// TIA Portal project "Bekletme_Kesmesi_Uygulaması_V1" (V16)
// Vorlageprojekt für das Buch mit Zielsystem S7-1200

(* hardware
DEVICE "S7-1200-Station_1"  S7-1200 Station
   slot 0: "Baugruppenträger_0"  Rack  V1.0
   slot 1: "PLC_1"  CPU 1214C DC/DC/DC  6ES7 214-1AG40-0XB0  V4.4
*)

// ===== PLC "PLC_1"  CPU 1214C DC/DC/DC =====

VAR_GLOBAL   // PLC tag table "Standard-Variablentabelle"
   "Sistem_Start_Mem." AT %M10.0 : Bool;
   "Kenar_Darbesi_1" AT %M20.0 : Bool;
   "Alarm" AT %M30.0 : Bool;
   "Kenar_Darbesi_2" AT %M20.1 : Bool;
   "Tag_1" AT %MW32 : Word;
   "Tag_2" AT %MW34 : Int;
END_VAR

VAR_GLOBAL   // PLC tag table "İnput"
   "Start_But" AT %I0.0 : Bool;
   "Stop_But" AT %I0.1 : Bool;
   "Sürücü_Geri_Sensörü" AT %I0.2 : Bool;
   "Sürücü_İleri_Sensörü" AT %I0.3 : Bool;
   "Optik_Sensör" AT %I0.4 : Bool;
   "Konveyör_Hız_Ayarı" AT %IW30 : Int;
END_VAR

VAR_GLOBAL   // PLC tag table "Output"
   "Sürücü" AT %Q0.0 : Bool;
   "Uyarı_Lambası" AT %Q0.1 : Bool;
   "Konveyör_1" AT %QW30 : Int;
   "Konveyör_2" AT %QW32 : Int;
END_VAR

FUNCTION "MHJ-PLC-Lab-Function-S71200" : Void   // FC9000, SCL
{ S7_Optimized_Access := 'TRUE' }
VERSION : 0.1
   VAR_TEMP
      rdTimeReturn : Int;
      outputTime : DTL;
      SyncVal : Byte;
      forVal : Int;
      forVal_2 : Int;
      Value : Byte;
   END_VAR
   VAR CONSTANT
      CompVal : Byte := 16#34;
      Value_01 : Byte := 16#11;
      Value_01_DW : DWord := 16#A165_D992;
      Value_02_DW : DWord := 16#58BE_4401;
   END_VAR
BEGIN

   #Value:=PEEK(area := 16#82,
        dbNumber := 0,
        byteOffset := 511);
   #Value := #Value + 1;

   POKE(area := 16#82,
        dbNumber := 0,
        byteOffset := 511,
        value := #Value);

   POKE(area:=16#81,
        dbNumber:=0,
        byteOffset:=1016,
        value:=#Value_01_DW);
   POKE(area := 16#81,
        dbNumber := 0,
        byteOffset := 1020,
        value := #Value_02_DW);

   POKE(area := 16#81,
        dbNumber := 0,
        byteOffset := 511,
        value := B#16#00);

   FOR #forVal := 0 TO 120 DO
       FOR #forVal_2:=0 TO 10 DO
           #rdTimeReturn:=RD_SYS_T(#outputTime);
           #rdTimeReturn := WR_SYS_T(#outputTime);
           #rdTimeReturn := RD_SYS_T(#outputTime);
           #rdTimeReturn := WR_SYS_T(#outputTime);
       END_FOR;
       #SyncVal:= PEEK(area := 16#81,
                      dbNumber := 0,
                      byteOffset := 511);
       IF #SyncVal = #CompVal THEN
          GOTO M_1;
       END_IF;
   END_FOR;
   RETURN;

   M_1:
   POKE(area := 16#81,
        dbNumber := 0,
        byteOffset := 511,
        value := B#16#0);
END_FUNCTION

ORGANIZATION_BLOCK "Main"   // OB1, LAD, ProgramCycle
TITLE = "Main Program Sweep (Cycle)"
{ S7_Optimized_Access := 'TRUE' }
VERSION : 0.1
   VAR_INPUT
      Initial_Call : Bool;   // Initial call of this OB
      Remanence : Bool;   // =True, if remanent data are available
   END_VAR
   VAR_TEMP   // added for the SCL form of the ladder/FBD networks
      _w1 : Bool;
   END_VAR
BEGIN

REGION Network 1: Konnektierungsbaustein für PLC-Lab
   // Im Netzwerk 1 wird der Konnektierungsbaustein für PLC-Lab aufgerufen.
   // Dieser Aufruf darf nicht entfernt werden!
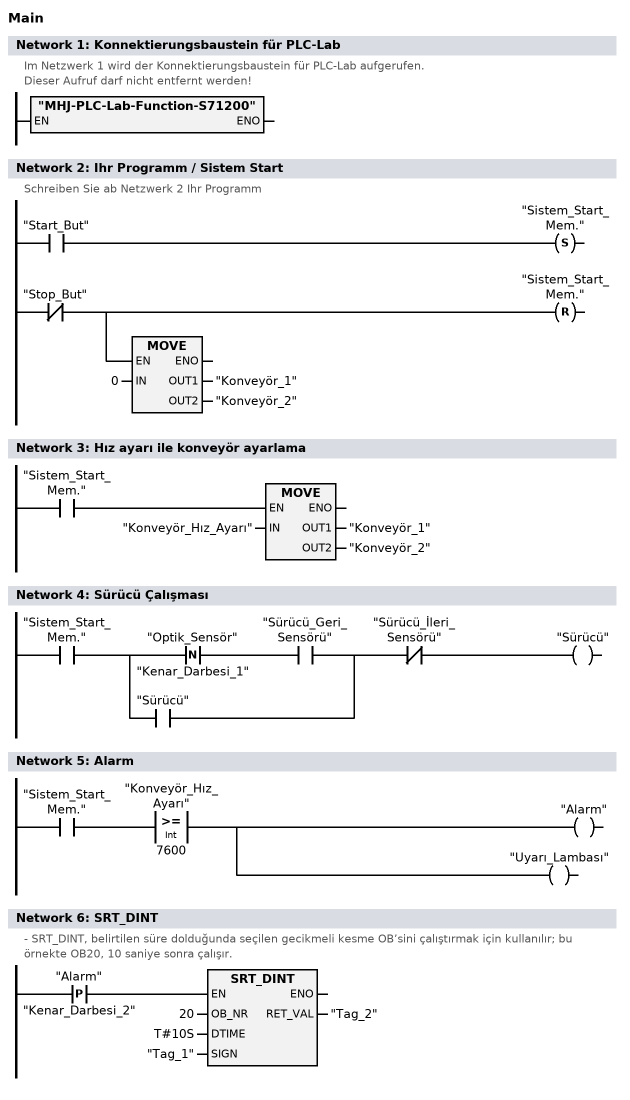
   RUNG wire#powerrail
      "MHJ-PLC-Lab-Function-S71200"()
   END_RUNG
   // the same network as SCL:
   "MHJ-PLC-Lab-Function-S71200"();
END_REGION

REGION Network 2: Ihr Programm / Sistem Start
   // Schreiben Sie ab Netzwerk 2 Ihr Programm
   RUNG wire#powerrail
      Contact( "Start_But" )
      S_Coil( "Sistem_Start_Mem." )
   END_RUNG
   RUNG wire#powerrail
      I_Contact( "Stop_But" )
      wire#w1
      R_Coil( "Sistem_Start_Mem." )
   END_RUNG
   RUNG wire#w1
      Move(in := 0, out1 => "Konveyör_1", out2 => "Konveyör_2")
   END_RUNG
   // the same network as SCL:
   IF "Start_But" THEN "Sistem_Start_Mem." := TRUE; END_IF;
   IF NOT "Stop_But" THEN
       "Sistem_Start_Mem." := FALSE;
       "Konveyör_1" := 0;
       "Konveyör_2" := 0;
   END_IF;
END_REGION

REGION Network 3: Hız ayarı ile konveyör ayarlama
   RUNG wire#powerrail
      Contact( "Sistem_Start_Mem." )
      Move(in := "Konveyör_Hız_Ayarı", out1 => "Konveyör_1", out2 => "Konveyör_2")
   END_RUNG
   // the same network as SCL:
   IF "Sistem_Start_Mem." THEN
       "Konveyör_1" := "Konveyör_Hız_Ayarı";
       "Konveyör_2" := "Konveyör_Hız_Ayarı";
   END_IF;
END_REGION

REGION Network 4: Sürücü Çalışması
   RUNG wire#powerrail
      Contact( "Sistem_Start_Mem." )
      wire#w1
      N_Contact(operand := "Optik_Sensör", bit := "Kenar_Darbesi_1")
      Contact( "Sürücü_Geri_Sensörü" )
      wire#w2
      I_Contact( "Sürücü_İleri_Sensörü" )
      Coil( "Sürücü" )
   END_RUNG
   RUNG wire#w1
      Contact( "Sürücü" )
   END_RUNG wire#w2
   // the same network as SCL:
   #_w1 := "Sistem_Start_Mem." AND NOT "Optik_Sensör" AND "Kenar_Darbesi_1";   // falling edge of "Optik_Sensör"
   "Kenar_Darbesi_1" := "Optik_Sensör";
   "Sürücü" := ((#_w1 AND "Sürücü_Geri_Sensörü") OR ("Sistem_Start_Mem." AND "Sürücü")) AND NOT "Sürücü_İleri_Sensörü";
END_REGION

REGION Network 5: Alarm
   RUNG wire#powerrail
      Contact( "Sistem_Start_Mem." )
      { S7_Templates := "SrcType := Int" } GE_Contact(in1 := "Konveyör_Hız_Ayarı", in2 := 7600)
      wire#w1
      Coil( "Alarm" )
   END_RUNG
   RUNG wire#w1
      Coil( "Uyarı_Lambası" )
   END_RUNG
   // the same network as SCL:
   "Alarm" := "Sistem_Start_Mem." AND ("Konveyör_Hız_Ayarı" >= 7600);
   "Uyarı_Lambası" := "Alarm";
END_REGION

REGION Network 6: SRT_DINT
   // - SRT_DINT, belirtilen süre dolduğunda seçilen gecikmeli kesme OB’sini çalıştırmak için kullanılır; bu örnekte OB20, 10 saniye sonra çalışır.
   #_w1 := "Alarm" AND NOT "Kenar_Darbesi_2";   // rising edge of "Alarm"
   "Kenar_Darbesi_2" := "Alarm";
   IF #_w1 THEN "Tag_2" := SRT_DINT(OB_NR := 20, DTIME := T#10S, SIGN := "Tag_1"); END_IF;
END_REGION
END_ORGANIZATION_BLOCK

ORGANIZATION_BLOCK "Sistem Trig"   // OB20, LAD, TimeDelayInterrupt
{ S7_Optimized_Access := 'TRUE' }
VERSION : 0.1
   VAR_INPUT
      Sign : Word;   // Identifier input (SIGN) passed to triggering call of SRT_DINT
   END_VAR
BEGIN

REGION Network 1: Sistem Trig
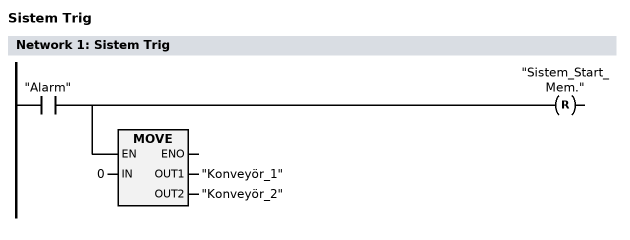
   RUNG wire#powerrail
      Contact( "Alarm" )
      wire#w1
      R_Coil( "Sistem_Start_Mem." )
   END_RUNG
   RUNG wire#w1
      Move(in := 0, out1 => "Konveyör_1", out2 => "Konveyör_2")
   END_RUNG
   // the same network as SCL:
   IF "Alarm" THEN
       "Sistem_Start_Mem." := FALSE;
       "Konveyör_1" := 0;
       "Konveyör_2" := 0;
   END_IF;
END_REGION
END_ORGANIZATION_BLOCK